FUNCTION alg_M_Distributing_a_Dstopled : BOOL
VAR_INPUT
	state: STATE;
END_VAR

alg_M_Distributing_a_Dstopled := (((((((state.dvar_M_Distributing) <> (elit_wait_start)) AND ((state.dvar_M_Distributing) <> (elit_init2))) AND ((state.dvar_M_Distributing) <> (elit_droppoint))) AND ((state.dvar_M_Distributing) <> (elit_movetopickup))) AND ((state.dvar_M_Distributing) <> (elit_down))) AND ((state.dvar_M_Distributing) <> (elit_gopickup))) AND ((state.dvar_M_Distributing) <> (elit_goback));

END_FUNCTION

(* stored: Version 1.1.0.1, ProductVersion 3.1.4022.18
   POU alg_M_Distributing_a_Dstopled: Id {3328c36d-1f45-4931-92e8-8e764f8e17cf}, SpecialFunc None *)
